// Interface with properties only.
INTERFACE I_WithRPC

// A method with all types of input and outputs as well as a return type.
{attribute 'TcRpcEnable'}
METHOD FullMethod : UDINT
VAR_INPUT
	InArg1  	: STRING(64);
	InArg2		: Tc2_System.ST_CpuCoreInfo; 
END_VAR
VAR_IN_OUT
	InOutArg1	: POINTER TO __UXINT;
END_VAR
VAR_OUTPUT
	OutArg1		: Tc2_System.E_SeekOrigin;
	OutArg2		: Tc2_System.T_MaxString;
END_VAR
END_METHOD

// First property.
{attribute 'TcRpcEnable'}
PROPERTY Prop1 : BOOL
GET
END_GET
SET
END_SET
END_PROPERTY

// A method that has no arguments.
{attribute 'TcRpcEnable'}
METHOD VoidMethod
VAR_INPUT
END_VAR
END_METHOD

END_INTERFACE

(* stored: Version 1.1.0.1, ProductVersion 3.1.4024.15
   Itf I_WithRPC: Id {d350ebc8-e31d-4308-ba70-8a44e5172862}
   Method FullMethod: Id {36f4f363-fa2c-4d5b-bdc2-ee918a8a3ce2}
   Property Prop1: Id {fe69b81d-a312-439d-ae8d-c7ae23a3b0f0}
   Get Get: Id {7c78c44b-2766-4f43-ac24-51ed4701ff11}
   Set Set: Id {443fe1ce-a341-4232-bb90-b58dd34a4d85}
   Method VoidMethod: Id {ef34f1b7-1f76-4a5f-841b-e4533169acd2} *)
